(* CoDeSys 2.3.9.50 project: XC152_profibusXNE2cnt_237SP7.pro *)
(* Libraries: Standard.lib 5.4.06 14:34:00, Util.lib 20.3.15 10:30:08, SysLibCallback.lib 28.12.11 14:04:40, SysLibSockets.lib 7.5.14 08:02:16, SysLibTasks.lib 28.12.11 14:04:40, SysLibRtc.lib 28.12.11 14:04:40, SysLibFile.lib 28.12.11 14:04:40, SysLibPlcCtrl.lib 28.12.11 14:04:40 *)

(* POU PLC_PRG, ST *)
PROGRAM PLC_PRG
VAR
	Control_A1: BYTE;
	diCounterValue1: DINT;
END_VAR
%QB0 := Control_A1;

%IB0;
%IB1;
%IB2;
%IB3;
%IB4;
%IB5;
%IB6;
%IB7;
%IB8;
%IB9;
%IB10;
%IB11;
%IB12;
%IB13;
%IB14;
%IB15;
(* Pour avoir une valeur de comptage qui s'incremente, une negation a été nécessaire*)
diCounterValue1:= -  (UDINT_TO_DINT((BYTE_TO_UDINT(%IB12)*16777216)+(BYTE_TO_UDINT(%IB13)*65536)+(BYTE_TO_UDINT(%IB14)*256)+BYTE_TO_UDINT(%IB15)));
END_PROGRAM

(* Visualisation MAPAGE
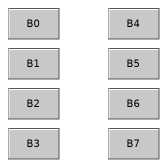
button at (10,10)-(61,41): text "B0"; toggles PLC_PRG.Control_A1.0
button at (110,10)-(161,41): text "B4"; toggles PLC_PRG.Control_A1.4
button at (10,50)-(61,81): text "B1"; toggles PLC_PRG.Control_A1.1
button at (10,90)-(61,121): text "B2"; toggles PLC_PRG.Control_A1.2
button at (10,130)-(61,161): text "B3"; toggles PLC_PRG.Control_A1.3
button at (110,50)-(161,81): text "B5"; toggles PLC_PRG.Control_A1.5
button at (110,90)-(161,121): text "B6"; toggles PLC_PRG.Control_A1.6
button at (110,130)-(161,161): text "B7"; toggles PLC_PRG.Control_A1.7
*)
